// TIA Portal V16 export
// export: Created 2020-12-17T10:21:04.2144047Z, ExportSetting WithDefaults, DisplayName Totally Integrated Automation Portal, DisplayVersion V16 Update 2, DisplayName TIA Portal Version Control Interface, DisplayVersion V16 Update 2, DisplayName TIA Portal Openness, DisplayVersion V16 Update 2, DisplayName STEP 7 Professional, DisplayVersion V16 Update 2, DisplayName STEP 7 Safety, DisplayVersion V16, DisplayName WinCC Advanced / Unified PC, DisplayVersion V16 Update 2
FUNCTION "Block_L1" : Void   // FC1, LAD
{ S7_Optimized_Access := 'TRUE' }
VERSION : 0.1
// stored: AutoNumber true, IsIECCheckEnabled false, SetENOAutomatically false, UDAEnableTagReadback false
   VAR_TEMP
      Tag_1 : Bool;
      Tag_2 : Bool;
   END_VAR
BEGIN

REGION Network 1
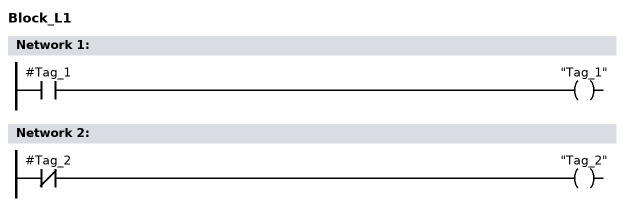
   RUNG wire#powerrail
      Contact( #Tag_1 )
      Coil( "Tag_1" )
   END_RUNG
   // the same network as SCL:
   "Tag_1" := #Tag_1;
END_REGION

REGION Network 2
   RUNG wire#powerrail
      I_Contact( #Tag_2 )
      Coil( "Tag_2" )
   END_RUNG
   // the same network as SCL:
   "Tag_2" := NOT #Tag_2;
END_REGION
END_FUNCTION
